{attribute 'qualified_only'}
VAR_GLOBAL
	iIloscZdefiniowanychZdarzen				: INT := 0;
	
END_VAR

(* stored: Version 1.1.0.1, ProductVersion 3.1.4024.11
   GVL ObslugaAlarmow_Zmienne: Id {5f0d00b4-0efa-4995-a0b3-b4e66e0f7bc4} *)
